FUNCTION_BLOCK XtsMotorModule EXTENDS CyclicBase
VAR
	MyModuleIoInterface : I_TcIoXtsPartModule;
	MyModuleCoEInterface : I_AT2xxxXtsMotor;
	CurrentLive: DINT;
	MaxCurrent: DINT;
	Nominal24Vdc : LREAL := 24000;
	Nominal48Vdc : LREAL := 48000;
	InSim : BOOL;
	Module24Vdc: UINT;
	Module48Vdc: UINT;
END_VAR

METHOD PUBLIC  Cycle : HRESULT
VAR_INPUT
END_VAR
IF MyModuleCoEInterface <> 0 AND NOT InSim THEN
	MyModuleCoEInterface.InfoData.Update();
	MyModuleCoEInterface.DiagData.Update();
	//MyModuleCoEInterface.AllCoE.UpdateAllCoEData();
	CurrentLive:=MyModuleCoEInterface.InfoData.OverallCurrent;
	MaxCurrent:=MyModuleCoEInterface.InfoData.MaxOverallCurrentLast500ms;
	Module24Vdc := MyModuleCoEInterface.InfoData.AuxiliaryVoltage24V;
	Module48Vdc := MyModuleCoEInterface.InfoData.DcLinkVoltage;
END_IF
END_METHOD

METHOD Initialise : HRESULT
VAR_INPUT
END_VAR
IF MyModuleIoInterface.P_IsInitialized THEN
	Initialise := 2;
END_IF
END_METHOD

METHOD Is24VOK : HRESULT
VAR_INPUT
END_VAR
IF MyModuleCoEInterface.InfoData.AuxiliaryVoltage24V < (Nominal24Vdc * 0.9) THEN
	Is24VOK := 1;
END_IF
IF MyModuleCoEInterface.InfoData.AuxiliaryVoltage24V > (Nominal24Vdc * 1.1) THEN
	Is24VOK := 1;
END_IF
END_METHOD

METHOD Is48VOK : HRESULT
VAR_INPUT
END_VAR
IF MyModuleCoEInterface.InfoData.DcLinkVoltage < (Nominal48Vdc * 0.9) THEN
	Is48VOK := 1;
END_IF
IF MyModuleCoEInterface.InfoData.DcLinkVoltage > (Nominal48Vdc * 1.1) THEN
	Is48VOK := 1;
END_IF
END_METHOD

PROPERTY MyCoEInterface : I_AT2xxxXtsMotor
GET
MyCoEInterface := MyModuleCoEInterface;
END_GET
SET
MyModuleCoEInterface := MyCoEInterface;
END_SET
END_PROPERTY

PROPERTY MyModuleInterface : I_TcIoXtsPartModule
GET
MyModuleInterface := MyModuleIoInterface;
END_GET
SET
MyModuleIoInterface := MyModuleInterface;
END_SET
END_PROPERTY

METHOD SetInSim : HRESULT
VAR_INPUT
END_VAR
InSim := true;
END_METHOD

END_FUNCTION_BLOCK

(* stored: Version 1.1.0.1
   POU XtsMotorModule: Id {447db564-ab24-433c-b078-4cedd1c7411e}, SpecialFunc None
   Method Cycle: Id {1188f197-bbd0-4970-903a-af249f1ed9e0}
   Method Initialise: Id {0d230f78-299f-458d-bcac-a537a1290197}
   Method Is24VOK: Id {9b08696d-e0e1-46f9-950f-7b12a84e7180}
   Method Is48VOK: Id {f76f25e2-8796-412c-b16e-72d1b643b91d}
   Property MyCoEInterface: Id {deb7d555-7556-4b66-ad9b-3c26c6b34c42}
   Get Get: Id {8461ccf8-f83e-404c-a347-71da6ba8563a}
   Set Set: Id {e0b2dbb9-69f1-4a7b-955f-87ac0078a8d2}
   Property MyModuleInterface: Id {2168d719-80a8-412e-a875-7c102bb8a0d2}
   Get Get: Id {89cf633f-414b-41a7-b6da-6e0666d662cd}
   Set Set: Id {c9ca3467-a5fd-4003-89ce-a9baa660bd96}
   Method SetInSim: Id {13eee03f-0b41-4595-95d5-55a5ef2b6f3f} *)
